PROGRAM P_ReadSesnors
VAR
	fbReadAcc : FB_ReadAccelerometer;
	
	accX AT %Q* : LREAL;
	accY AT %Q* : LREAL;
	accZ AT %Q* : LREAL;
END_VAR

fbReadAcc(accX=>accX, accY=>accY, accZ=>accZ);

END_PROGRAM

(* stored: Version 1.1.0.1, ProductVersion 3.1.4024.13
   POU P_ReadSesnors: Id {e83dad1a-1bca-4649-aeed-6950f3612e99}, SpecialFunc None *)
